TYPE ST_Safety_get :
STRUCT
	b_SafetyOK					: BOOL;
	b_EstopChannelAOK			: BOOL;		
	b_EstopChannelBOK			: BOOL;		
	b_InsulationMonitorOK		: BOOL;	
	b_MRCDBOK					: BOOL;	
	b_InverterDoorOK            : BOOL;
	b_ZptOK				        : BOOL;
END_STRUCT
END_TYPE

(* stored: Version 1.1.0.1, ProductVersion 3.1.4024.12
   DUT ST_Safety_get: Id {718e49dc-7a62-48d6-bebd-68c0d0bcdfdf} *)
